SUBAPPLICATION Uebung_205b (* Interlock: ILOCK_SWITCH_PROTECT (Motor Reversierung Priorität mit Schutzzeit) *)
  (* Standard: 61499-2; Description: Copyright (c) 2023 Meisterschulen am Ostbahnhof This program and the accompanying materials are made available under the terms of the Eclipse Public License 2.0 which is available at https://www.eclipse.org/legal/epl-2.0/ SPDX-License-Identifier: EPL-2.0 *)
  (* Version 1.0, 2026-04-19, Franz Höpfinger, Meisterschulen am Ostbahnhof, initial API and implementation and/or initial documentation *)
  PACKAGE Uebungen;
  IMPORT logiBUS::io::DI::logiBUS_DI::Input_I1;
  IMPORT logiBUS::io::DI::logiBUS_DI::Input_I2;
  IMPORT logiBUS::io::DQ::logiBUS_DO::Output_Q5;
  IMPORT logiBUS::io::DQ::logiBUS_DO::Output_Q6;
  IMPORT logiBUS::io::DQ::logiBUS_DO::Output_Q56;
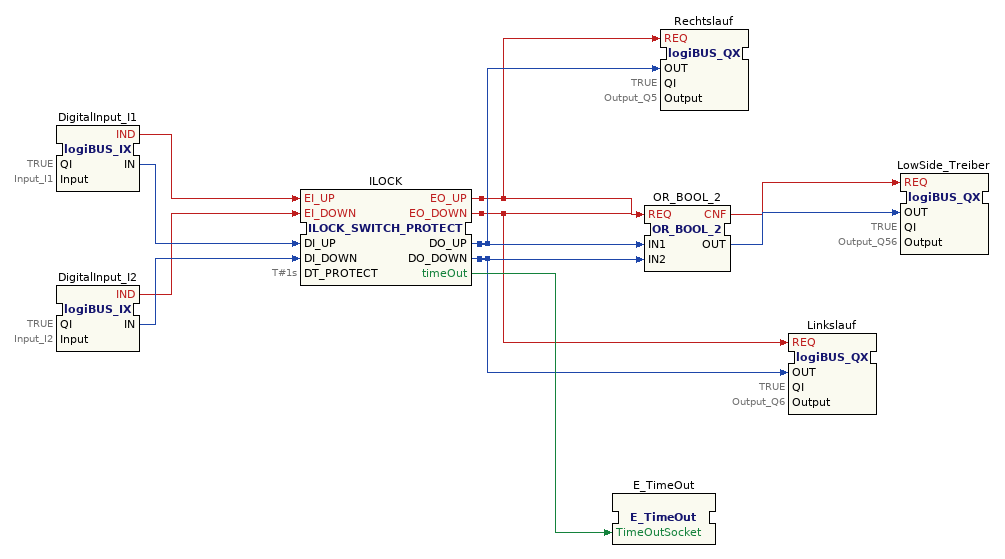
  FBS
    DigitalInput_I1 : logiBUS::io::DI::logiBUS_IX(QI := TRUE, Input := Input_I1);
    DigitalInput_I2 : logiBUS::io::DI::logiBUS_IX(QI := TRUE, Input := Input_I2);
    ILOCK : logiBUS::signalprocessing::interlock::ILOCK_SWITCH_PROTECT(DT_PROTECT := T#1s);
    Rechtslauf : logiBUS::io::DQ::logiBUS_QX(QI := TRUE, Output := Output_Q5);
    Linkslauf : logiBUS::io::DQ::logiBUS_QX(QI := TRUE, Output := Output_Q6);
    LowSide_Treiber : logiBUS::io::DQ::logiBUS_QX(QI := TRUE, Output := Output_Q56);
    OR_BOOL_2 : iec61131::booleanOperators::OR_BOOL_2;
    E_TimeOut : iec61499::events::E_TimeOut;
  END_FBS
  EVENT_CONNECTIONS
    DigitalInput_I1.IND TO ILOCK.EI_UP;
    DigitalInput_I2.IND TO ILOCK.EI_DOWN;
    ILOCK.EO_UP TO Rechtslauf.REQ;
    ILOCK.EO_DOWN TO Linkslauf.REQ;
    ILOCK.EO_UP TO OR_BOOL_2.REQ;
    ILOCK.EO_DOWN TO OR_BOOL_2.REQ;
    OR_BOOL_2.CNF TO LowSide_Treiber.REQ;
  END_CONNECTIONS
  DATA_CONNECTIONS
    DigitalInput_I1.IN TO ILOCK.DI_UP;
    DigitalInput_I2.IN TO ILOCK.DI_DOWN;
    ILOCK.DO_UP TO Rechtslauf.OUT;
    ILOCK.DO_DOWN TO Linkslauf.OUT;
    ILOCK.DO_UP TO OR_BOOL_2.IN1;
    ILOCK.DO_DOWN TO OR_BOOL_2.IN2;
    OR_BOOL_2.OUT TO LowSide_Treiber.OUT;
  END_CONNECTIONS
  ADAPTER_CONNECTIONS
    ILOCK.timeOut TO E_TimeOut.TimeOutSocket;
  END_CONNECTIONS
END_SUBAPPLICATION
